ABB RAPID module: TCPZ_tool_jnj1.MOD

MODULE TCPZ_tool_jnj1
	! Points are read in order of declaration.
  ! Please do not change the order of points!

  LOCAL PERS robtarget pTCPZ_Point1:=[[462.1133,187.2552,210.3063],[0.516728281974792,-0.123953819274902,0.813863039016724,0.235062226653099],[0,-1,0,1],[9E+09,9E+09,9E+09,9E+09,9E+09,9E+09]];
	LOCAL PERS robtarget pTCPZ_Point2:=[[429.3243,181.4934,193.4006],[0.505189120769501,0.385440737009048,0.756630182266235,0.15404599905014],[0,0,0,1],[9E+09,9E+09,9E+09,9E+09,9E+09,9E+09]];
	LOCAL PERS robtarget pTCPZ_Point3:=[[455.4832,221.7342,219.5257],[0.402685135602951,-0.698162615299225,0.549405992031097,0.220378428697586],[0,-1,0,1],[9E+09,9E+09,9E+09,9E+09,9E+09,9E+09]];
	LOCAL PERS robtarget pTCPZ_Point4:=[[431.0109,218.4641,209.1816],[0.433560401201248,-0.77957159280777,0.426138877868652,0.150662273168564],[0,-1,-1,1],[9E+09,9E+09,9E+09,9E+09,9E+09,9E+09]];
	LOCAL PERS robtarget pTCPZ_ElongZ:=[[457.6317,198.0575,214.7151],[0.52157986164093,-0.451503098011017,0.679097175598145,0.25085124373436],[0,-1,0,1],[9E+09,9E+09,9E+09,9E+09,9E+09,9E+09]];

ENDMODULE
